// This function has been automatically generated from the project information.
{attribute 'signature_flag' := '1073741824'}
{attribute 'TcGenerated'}
{attribute 'no-analysis'}
FUNCTION F_GetTitle : WSTRING
VAR_INPUT
	
END_VAR

F_GetTitle := "CNM Production Metrics";

END_FUNCTION

(* stored: Version 1.1.0.1
   POU F_GetTitle: Id {98c661c6-0d6f-495f-9237-bc36e3c08fcf}, SpecialFunc None *)
